Staubli VAL3: JPOINT.dtx

public TrajJoint tTraj{}
